ABB RobotStudio station: ProjectAPM.rsstnx

Station ProjectAPM (saved by RobotStudio 26.2.11700.0)
Controller Controller460, task T_ROB1: task frame (RAPID world) sits at (200, 0, 1400) mm in the station
Controller Controller460
  mechanical unit ROB_1: IRB460_110_240__01, 6 joints, base frame (0, 0, 0) mm
Layout (positions relative to the parent item):
  - IRB460_110_240__01 [mechanism, from %ABB.RobotStudio.Models.IRB460%\IRB460_110_240__02.rslib] at (200, 0, 1400) mm; joint values [-0.2198, 0.4757, -0.3433, 0.02] (rad or m)
  - SC_PM_PLC [smart component, from %AD3BFF28-CFC8-4A83-9FC3-1BF366785115%\SC_PM_PLC.rslib]
      properties: SimulationQuickStart=; StatisticsInfo=; con0_ID={755c8d52-c703-4704-be43-8eb584e27281}; con0_pmPLC_dpSelectedFlowID=; con0_T_ROB1_ID={f23f62ef-cbdf-4f0c-95f8-80ade90c0930}; con0_T_ROB1_ObjectReleased=(none)
  - PalletDispenser 1300_1300_300 [smart component, from %567FE6EA-F242-46D1-87E8-57A1ECE2G0DC%\PalletDispenser 1300_1300_300.rslib] at (2250, -5860, 70) mm, rotated rx 0 ry 0 rz 90 deg
      properties: PreparationTime_ToPick=0; Product_ToPick=; ClearTime_Placed=0; Product_Placed=
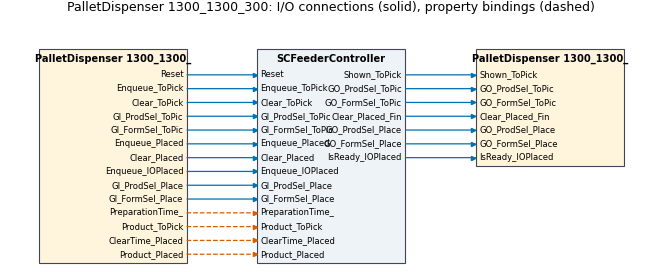
      connections:
        PalletDispenser 1300_1300_300.Reset -> SCFeederController.Reset
        PalletDispenser 1300_1300_300.Enqueue_ToPick -> SCFeederController.Enqueue_ToPick
        SCFeederController.Shown_ToPick -> PalletDispenser 1300_1300_300.Shown_ToPick
        PalletDispenser 1300_1300_300.Clear_ToPick -> SCFeederController.Clear_ToPick
        PalletDispenser 1300_1300_300.GI_ProdSel_ToPick -> SCFeederController.GI_ProdSel_ToPick
        PalletDispenser 1300_1300_300.GI_FormSel_ToPick -> SCFeederController.GI_FormSel_ToPick
        SCFeederController.GO_ProdSel_ToPick -> PalletDispenser 1300_1300_300.GO_ProdSel_ToPick
        SCFeederController.GO_FormSel_ToPick -> PalletDispenser 1300_1300_300.GO_FormSel_ToPick
        SCFeederController.Clear_Placed_Finished -> PalletDispenser 1300_1300_300.Clear_Placed_Finished
        PalletDispenser 1300_1300_300.Enqueue_Placed -> SCFeederController.Enqueue_Placed
        PalletDispenser 1300_1300_300.Clear_Placed -> SCFeederController.Clear_Placed
        PalletDispenser 1300_1300_300.Enqueue_IOPlacedRequest -> SCFeederController.Enqueue_IOPlacedRequest
        PalletDispenser 1300_1300_300.GI_ProdSel_PlacedRequest -> SCFeederController.GI_ProdSel_PlacedRequest
        PalletDispenser 1300_1300_300.GI_FormSel_PlacedRequest -> SCFeederController.GI_FormSel_PlacedRequest
        SCFeederController.GO_ProdSel_PlacedRequest -> PalletDispenser 1300_1300_300.GO_ProdSel_PlacedRequest
        SCFeederController.GO_FormSel_PlacedRequest -> PalletDispenser 1300_1300_300.GO_FormSel_PlacedRequest
        SCFeederController.IsReady_IOPlacedRequest -> PalletDispenser 1300_1300_300.IsReady_IOPlacedRequest
        PalletDispenser 1300_1300_300.PreparationTime_ToPick => SCFeederController.PreparationTime_ToPick
        PalletDispenser 1300_1300_300.Product_ToPick => SCFeederController.Product_ToPick
        PalletDispenser 1300_1300_300.ClearTime_Placed => SCFeederController.ClearTime_Placed
        PalletDispenser 1300_1300_300.Product_Placed => SCFeederController.Product_Placed
    - PalletDispenser 1300_1300_300 [part, from %567FE6EA-F242-46D1-87E8-57A1ECE2G0DC%\PalletDispenser 1300_1300_300.rslib]
    - SCFeederController [smart component, from %AD3BFF28-CFC8-4A83-9FC3-1BF366785115%\SC_FeederController.rslib]
        properties: Product_Placed=12; ClearTime_Placed=0; PreparationTime_ToPick=0; Product_ToPick=12
  - SC_Conveyor600 [smart component]
  - SixPackComponent [smart component]
      signals: DI Start, DI Pieza, DO PosicionAg
      connections:
        Source_2.Executed -> LogicSRLatch.Set
        LogicSRLatch.Output -> LinearMover.Execute
        Source_3.Executed -> LogicSRLatch_2.Set
        LogicSRLatch_2.Output -> LinearMover.Execute
        LineSensor.SensorOut -> LogicGate.InputA
        SixPackComponent.Start -> LogicGate.InputB
        LogicGate.Output -> Source_3.Execute
        LineSensor.SensorOut -> Source_3.Execute
        LogicGate_2.Output -> Source_3.Execute
        SixPackComponent.Start -> LogicGate_4.InputA
        LogicGate_4.Output -> LogicGate_2.InputA
        SixPackComponent.Pieza -> LogicGate_4.InputB
        LogicGate_4.Output -> Source_3.Execute
        LineSensor_4.SensorOut -> LogicSRLatch_2.Reset
        SixPackComponent.Start -> Source_4.Execute
        Source_3.Copy => LinearMover.Object
    - SixPack [part] at (0, 3800, 165.66) mm, rotated rx 90 ry 0 rz 0 deg, size 377 x 385.4 x 237.4 mm
    - Conveyor_600 [smart component, from %567FE6EA-F242-46D1-87E8-57A1ECE2G0DC%\Conveyor_600.rslib] at (350, 1000, 0) mm, rotated rx 0 ry 0 rz 90 deg
        properties: PreparationTime_ToPick=0; Product_ToPick=; ClearTime_Placed=0; Product_Placed=
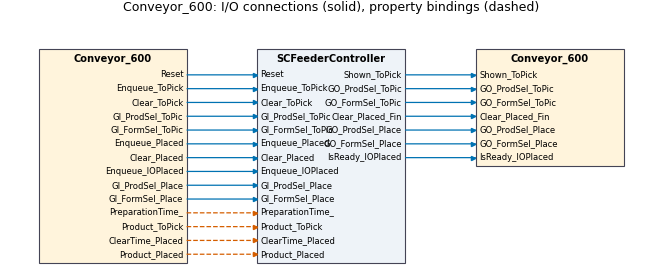
        connections:
          Conveyor_600.Reset -> SCFeederController.Reset
          Conveyor_600.Enqueue_ToPick -> SCFeederController.Enqueue_ToPick
          SCFeederController.Shown_ToPick -> Conveyor_600.Shown_ToPick
          Conveyor_600.Clear_ToPick -> SCFeederController.Clear_ToPick
          Conveyor_600.GI_ProdSel_ToPick -> SCFeederController.GI_ProdSel_ToPick
          Conveyor_600.GI_FormSel_ToPick -> SCFeederController.GI_FormSel_ToPick
          SCFeederController.GO_ProdSel_ToPick -> Conveyor_600.GO_ProdSel_ToPick
          SCFeederController.GO_FormSel_ToPick -> Conveyor_600.GO_FormSel_ToPick
          SCFeederController.Clear_Placed_Finished -> Conveyor_600.Clear_Placed_Finished
          Conveyor_600.Enqueue_Placed -> SCFeederController.Enqueue_Placed
          Conveyor_600.Clear_Placed -> SCFeederController.Clear_Placed
          Conveyor_600.Enqueue_IOPlacedRequest -> SCFeederController.Enqueue_IOPlacedRequest
          Conveyor_600.GI_ProdSel_PlacedRequest -> SCFeederController.GI_ProdSel_PlacedRequest
          Conveyor_600.GI_FormSel_PlacedRequest -> SCFeederController.GI_FormSel_PlacedRequest
          SCFeederController.GO_ProdSel_PlacedRequest -> Conveyor_600.GO_ProdSel_PlacedRequest
          SCFeederController.GO_FormSel_PlacedRequest -> Conveyor_600.GO_FormSel_PlacedRequest
          SCFeederController.IsReady_IOPlacedRequest -> Conveyor_600.IsReady_IOPlacedRequest
          Conveyor_600.PreparationTime_ToPick => SCFeederController.PreparationTime_ToPick
          Conveyor_600.Product_ToPick => SCFeederController.Product_ToPick
          Conveyor_600.ClearTime_Placed => SCFeederController.ClearTime_Placed
          Conveyor_600.Product_Placed => SCFeederController.Product_Placed
      - 600_guide [part, from %567FE6EA-F242-46D1-87E8-57A1ECE2G0DC%\Conveyor_600.rslib]
      - SCFeederController [smart component, from %AD3BFF28-CFC8-4A83-9FC3-1BF366785115%\SC_FeederController.rslib]
          properties: Product_Placed=; ClearTime_Placed=0; PreparationTime_ToPick=0; Product_ToPick=
    - LinearMover [smart component, from Components\LinearMover.rslib]
        properties: Object=(none); Direction=[0 -1 0]; Speed=5; Reference=Global; ReferenceObject=(none)
    - Source_3 [smart component, from Components\Source.rslib]
        properties: Source=SixPack; Copy=(none); Parent=(none); Position=[0 3.8000000000000003 0.96]; Orientation=[1.5707963267948966 -0 0]; Transient=true; PhysicsBehavior=0
    - LogicSRLatch_2 [smart component, from Components\LogicSRLatch.rslib]
    - LineSensor_4 [smart component, from Components\LineSensor.rslib]
        properties: Start=[0.35000000000000003 1.3 0.85]; End=[-0.29 1.3 0.85]; Length=0.64; Radius=0; Tag=(none); SenseMultiple=false; SensedPart=(none); SensedPoint=[0 0 0]
      - _sensorPart_ [part], size 640 x 0 x 0 mm
    - LogicGate_4 [smart component, from Components\LogicGate.rslib]
        properties: Operator=OR; Delay=0
    - Source_4 [smart component, from Components\Source.rslib]
        properties: Source=slipSheet; Copy=(none); Parent=(none); Position=[-1.3 -2 0.4]; Orientation=[0 0 0]; Transient=true; PhysicsBehavior=0
    - SixPack_65 [part] at (0, 3800, 960) mm, rotated rx 90 ry 0 rz 0 deg, size 377 x 385.4 x 237.4 mm
    - SixPack_171 [part] at (0, 3800, 960) mm, rotated rx 90 ry 0 rz 0 deg, size 377 x 385.4 x 237.4 mm
    - SixPack_349 [part] at (0, 3800, 960) mm, rotated rx 90 ry 0 rz 0 deg, size 377 x 385.4 x 237.4 mm
  - Grashping [smart component]
      signals: DI Atach, DI Detatch
      connections:
        LineSensor_10.SensorOut -> Attacher.Execute
        Grashping.Atach -> LogicGate_3.InputA
        LogicGate_3.Output -> Detacher.Execute
        Grashping.Atach -> LineSensor_10.Active
        Grashping.Detatch -> Detacher.Execute
        Grashping.Atach -> LineSensor_11.Active
        LineSensor_11.SensorOut -> Attacher.Execute
        Grashping.Detatch -> Attacher_2.Execute
        Grashping.Detatch -> LineSensor_3.Active
        LineSensor_10.SensedPart => Attacher.Child
        Attacher.Child => Detacher.Child
        LineSensor_11.SensedPart => Attacher.Child
        Attacher.Child => Attacher_2.Child
        LineSensor_3.SensedPart => Attacher_2.Parent
    - Attacher [smart component, from Components\Attacher.rslib]
        properties: Parent=ClampOneZoneGripper; Flange=0; Child=(none); Mount=false; Offset=[0 0 0]; Orientation=[0 0 0]
    - Detacher [smart component, from Components\Detacher.rslib]
        properties: Child=(none); KeepPosition=true
    - ClampOneZoneGripper [smart component, from %8E81373A-26AF-41AD-988A-D568DD9CCF0C%\ClampOneZoneGripper.rslib] at (1705, 0, 2836) mm, rotated rx 180 ry 0 rz 180 deg
        properties: ReleasedObject=(none)
        connections:
          ClampOneZoneGripper.giOpenClamp -> Clamp1.giOpenClamp
          Clamp1.goClampOpened -> ClampOneZoneGripper.goClampOpened
          ClampOneZoneGripper.giOpenHook -> Clamp1.giOpenHook
          Clamp1.goHookOpened -> ClampOneZoneGripper.goHookOpened
          Clamp1.doObjectReleased -> Gripper_SCPropertiesMulti2Single.DI0
          Gripper_SCPropertiesMulti2Single.DO -> ClampOneZoneGripper.doObjectReleased
          Clamp1.ReleasedObject => Gripper_SCPropertiesMulti2Single.PI0
          Gripper_SCPropertiesMulti2Single.PO => ClampOneZoneGripper.ReleasedObject
      - ClampOneZoneGripper [mechanism, from %8E81373A-26AF-41AD-988A-D568DD9CCF0C%\ClampOneZoneGripper.rslib] at (0, 0, 0) mm; joint values [0.03, 0.085, -0.0436] (rad or m)
      - Clamp1 [smart component]
          properties: ReleasedObject=(none)
          signals: GI giOpenClamp, GO goClampOpened, GI giOpenHook, GO goHookOpened, DO doObjectReleased
          connections:
            Clamp1.giOpenClamp -> ClampControl.giOpenClamp
            ClampControl.goClampOpened -> Clamp1.goClampOpened
            Clamp1.giOpenHook -> HookControl.giOpenHook
            HookControl.goHookOpened -> Clamp1.goHookOpened
            ClampAct.doObjectDetached -> Clamp1.doObjectReleased
            ClampControl.Closed -> LogicSRLatch.Set
            ClampControl.Opening -> LogicSRLatch.Reset
            LogicSRLatch.Output -> ClampAct.diAttachOrDetach
            ClampControl.Closed -> LogicGate.InputA
            ClampControl.Opening -> LogicGate.InputB
            LogicGate.Output -> ClampAct.Active
            ClampAct.ReleasedObject => Clamp1.ReleasedObject
        - ClampControl [smart component]
            signals: GI giOpenClamp, GO goClampOpened, DO Closing, DO Closed, DO Opening, DO Opened
            connections:
              JointMoverClose.Executing -> ClampControl.Closing
              JointMoverClose.Executed -> ClampControl.Closed
              JointMoverOpen.Executing -> ClampControl.Opening
              JointMoverOpen.Executed -> ClampControl.Opened
              ClampControl.giOpenClamp -> MultiSignalJudgeOpen.GI0
              MultiSignalJudgeOpen.DO -> JointMoverOpen.Execute
              JointMoverOpen.Executed -> MultiSignalSetOpen.Set
              ClampControl.giOpenClamp -> MultiSignalJudgeClose.GI0
              MultiSignalJudgeClose.DO -> JointMoverClose.Execute
              JointMoverClose.Executed -> MultiSignalSetClose.Set
              MultiSignalSetOpen.Executed -> MutiSignalSelector.SelectorA
              MultiSignalSetOpen.GO0 -> MutiSignalSelector.GiA0
              MultiSignalSetClose.Executed -> MutiSignalSelector.SelectorB
              MultiSignalSetClose.GO0 -> MutiSignalSelector.GiB0
              MutiSignalSelector.goClampOpened -> ClampControl.goClampOpened
          - MultiSignalJudgeOpen [smart component, from %AD3BFF28-CFC8-4A83-9FC3-1BF366785115%\SC_MultiSignalJudge.rslib]
              properties: DICount=0; GICount=1
          - JointMoverOpen [smart component, from %AD3BFF28-CFC8-4A83-9FC3-1BF366785115%\SC_JointMoverEx.rslib]
              properties: Mechanism=ClampOneZoneGripper; Relative=false; Duration=0.2; UseJ1=false; J1=0; UseJ2=true; J2=0; UseJ3=false; J3=0
          - MultiSignalSetOpen [smart component, from %AD3BFF28-CFC8-4A83-9FC3-1BF366785115%\SC_MultiSignalSet.rslib]
              properties: DOCount=0; GOCount=1
          - MultiSignalJudgeClose [smart component, from %AD3BFF28-CFC8-4A83-9FC3-1BF366785115%\SC_MultiSignalJudge.rslib]
              properties: DICount=0; GICount=1
          - JointMoverClose [smart component, from %AD3BFF28-CFC8-4A83-9FC3-1BF366785115%\SC_JointMoverEx.rslib]
              properties: Mechanism=ClampOneZoneGripper; Relative=false; Duration=0.2; UseJ1=false; J1=0; UseJ2=true; J2=0.085; UseJ3=false; J3=0
          - MultiSignalSetClose [smart component, from %AD3BFF28-CFC8-4A83-9FC3-1BF366785115%\SC_MultiSignalSet.rslib]
              properties: DOCount=0; GOCount=1
          - MutiSignalSelector [smart component, from %AD3BFF28-CFC8-4A83-9FC3-1BF366785115%\SC_MultiSignalSelector.rslib]
              properties: DICountA=0; GICountA=1; DICountB=0; GICountB=1; PiGiA0=goClampOpened; PiGiB0=goClampOpened
        - HookControl [smart component]
            signals: GI giOpenHook, GO goHookOpened, DO Closing, DO Closed, DO Opening, DO Opened
            connections:
              JointMoverClose.Executing -> HookControl.Closing
              JointMoverClose.Executed -> HookControl.Closed
              JointMoverOpen.Executing -> HookControl.Opening
              JointMoverOpen.Executed -> HookControl.Opened
              HookControl.giOpenHook -> MultiSignalJudgeOpen.GI0
              MultiSignalJudgeOpen.DO -> JointMoverOpen.Execute
              JointMoverOpen.Executed -> MultiSignalSetOpen.Set
              HookControl.giOpenHook -> MultiSignalJudgeClose.GI0
              MultiSignalJudgeClose.DO -> JointMoverClose.Execute
              JointMoverClose.Executed -> MultiSignalSetClose.Set
              MultiSignalSetOpen.Executed -> MutiSignalSelector.SelectorA
              MultiSignalSetOpen.GO0 -> MutiSignalSelector.GiA0
              MultiSignalSetClose.Executed -> MutiSignalSelector.SelectorB
              MultiSignalSetClose.GO0 -> MutiSignalSelector.GiB0
              MutiSignalSelector.goHookOpened -> HookControl.goHookOpened
          - MultiSignalJudgeOpen [smart component, from %AD3BFF28-CFC8-4A83-9FC3-1BF366785115%\SC_MultiSignalJudge.rslib]
              properties: DICount=0; GICount=1
          - JointMoverOpen [smart component, from %AD3BFF28-CFC8-4A83-9FC3-1BF366785115%\SC_JointMoverEx.rslib]
              properties: Mechanism=ClampOneZoneGripper; Relative=false; Duration=0.2; UseJ1=false; J1=0; UseJ2=false; J2=0; UseJ3=true; J3=1.30899693899575
          - MultiSignalSetOpen [smart component, from %AD3BFF28-CFC8-4A83-9FC3-1BF366785115%\SC_MultiSignalSet.rslib]
              properties: DOCount=0; GOCount=1
          - MultiSignalJudgeClose [smart component, from %AD3BFF28-CFC8-4A83-9FC3-1BF366785115%\SC_MultiSignalJudge.rslib]
              properties: DICount=0; GICount=1
          - JointMoverClose [smart component, from %AD3BFF28-CFC8-4A83-9FC3-1BF366785115%\SC_JointMoverEx.rslib]
              properties: Mechanism=ClampOneZoneGripper; Relative=false; Duration=0.2; UseJ1=false; J1=0; UseJ2=false; J2=0; UseJ3=true; J3=-0.0436332312998582
          - MultiSignalSetClose [smart component, from %AD3BFF28-CFC8-4A83-9FC3-1BF366785115%\SC_MultiSignalSet.rslib]
              properties: DOCount=0; GOCount=1
          - MutiSignalSelector [smart component, from %AD3BFF28-CFC8-4A83-9FC3-1BF366785115%\SC_MultiSignalSelector.rslib]
              properties: DICountA=0; GICountA=1; DICountB=0; GICountB=1; PiGiA0=goHookOpened; PiGiB0=goHookOpened
        - ClampAct [smart component] at (0, 0, 323) mm
            properties: ReleasedObject=(none); AttachedObject=(none)
            signals: DI diAttachOrDetach, DI Active, DO doObjectAttached, DO doObjectDetached
            connections:
              ClampAct.diAttachOrDetach -> SC_VolumeGripper.AttachOrDetach
              SC_VolumeGripper.TriggerAttach -> Attacher.Execute
              SC_VolumeGripper.TriggerDetach -> Detacher.Execute
              Attacher.Executed -> ClampAct.doObjectAttached
              Detacher.Executed -> ClampAct.doObjectDetached
              ClampAct.Active -> SC_VolumeGripper.Active
              SC_VolumeGripper.AttachParent => Attacher.Parent
              SC_VolumeGripper.ChildToAttach => Attacher.Child
              SC_VolumeGripper.AttachedChild => Detacher.Child
              SC_VolumeGripper.AttachedChild => ClampAct.AttachedObject
              SC_VolumeGripper.ReleasedChild => ClampAct.ReleasedObject
          - SC_VolumeGripper [smart component, from %AD3BFF28-CFC8-4A83-9FC3-1BF366785115%\SC_VolumeGripper.rslib]
              properties: Position=[0 0 0]; Orientation=[0 0 0]; Size=[0.2 0.2 0.4]; AttachParent=ClampAct; ChildToAttach=(none); AttachedChild=(none); ReleasedChild=(none)
            - _sensorPart_ [part] at (-801.98, -408.83, 179.7) mm, rotated rx 0 ry 0 rz -55.45 deg, size 200 x 200 x 400 mm
          - Attacher [smart component, from Components\Attacher.rslib]
              properties: Parent=ClampAct; Flange=0; Child=(none); Mount=false; Offset=[0 0 0]; Orientation=[0 0 0]
          - Detacher [smart component, from Components\Detacher.rslib]
              properties: Child=(none); KeepPosition=true
        - LogicSRLatch [smart component, from Components\LogicSRLatch.rslib]
        - LogicGate [smart component, from Components\LogicGate.rslib]
            properties: Operator=OR; Delay=0
      - Gripper_SCPropertiesMulti2Single [smart component, from %AD3BFF28-CFC8-4A83-9FC3-1BF366785115%\SC_PropertiesMulti2Single.rslib]
          properties: Count=1; PO=(none); PI0=(none)
    - LineSensor_11 [smart component, from Components\LineSensor.rslib] at (1705, 0, 2309) mm, rotated rx 180 ry 0 rz 180 deg
        properties: Start=[1.5596846730803193E-09 -9.080824692198064E-08 1.1309381164892329E-07]; End=[1.5596846730803193E-09 -9.080824692198064E-08 -0.3109998869061883]; Length=0.31099999999999994; Radius=0.02; Tag=(none); SenseMultiple=false; SensedPart=(none); SensedPoint=[0.04999999237060547 1.3559327392578124 0.82682470703125]
      - _sensorPart_ [part], size 40 x 40 x 311 mm
    - Attacher_2 [smart component, from Components\Attacher.rslib]
        properties: Parent=DWPallet; Flange=0; Child=(none); Mount=false; Offset=[0 0 0]; Orientation=[0 0 0]
    - LineSensor_3 [smart component, from Components\LineSensor.rslib]
        properties: Start=[1.1362 -0.495618 0.43707799999999997]; End=[1.370596 -0.376168 0.532328]; Length=0.27978983150929543; Radius=0.003; Tag=(none); SenseMultiple=false; SensedPart=DWPallet; SensedPoint=[1.136199951171875 -0.4956180114746094 0.4370780029296875]
      - _sensorPart_ [part], size 237.7 x 124.8 x 100.9 mm
  - SixPack [graphiccomponentgroup] at (0, 0, -2383.34) mm
    - SixPack [part] at (150, 120, 0) mm, rotated rx 90 ry 0 rz 0 deg, size 238.9 x 259.1 x 149.8 mm
    - OuterLine [part], size 380 x 240 x 380 mm
    - Labels [part]
    - Origin [part], size 78.6 x 49.5 x 382.7 mm
  - PalletCoca [graphiccomponentgroup] at (900, -500, 450) mm
    - MainBody [part], size 2280 x 1000 x 150 mm
    - OuterLine [part], size 2280 x 1000 x 150 mm
    - Labels [part]
    - Origin [part], size 456.5 x 200.5 x 151 mm
  - Pallet [smart component]
      signals: DI Finish
      connections:
        Pallet.Finish -> LinearMover.Execute
        Pallet.Finish -> LinearMover2.Execute
        LinearMover2.Executed -> Sink.Execute
        Sink.Executed -> Positioner.Execute
        Pallet.Finish -> LineSensor.Active
        LinearMover2.Executed -> Source.Execute
        Pallet.Finish -> Timer.Active
        Timer.Output -> LineSensor_2.Active
        Pallet.Finish -> LogicSRLatch.Set
        LogicSRLatch.Output -> LineSensor_2.Active
        LineSensor_2.SensorOutPulse -> LogicSRLatch.Reset
        Pallet.Finish -> Timer.Active
        Timer.Output -> LineSensor_2.Active
        LinearMover2.Object => Sink.Object
        LineSensor.SensedPart => LinearMover2.Object
        LineSensor.SensedPart => Source.Source
        LineSensor_2.SensedPart => LinearMover2.Object
        LinearMover2.Object => Source.Source
    - LinearMover2 [smart component, from Components\LinearMover2.rslib]
        properties: Object=DWPallet; Direction=[1 0 0]; Distance=2.8000000000000003; Duration=5; Reference=Global; ReferenceObject=(none)
    - Source [smart component, from Components\Source.rslib]
        properties: Source=DWPallet; Copy=(none); Parent=(none); Position=[0.06 0.01 0.4]; Orientation=[0 0 0]; Transient=true; PhysicsBehavior=0
    - LineSensor_2 [smart component, from Components\LineSensor.rslib]
        properties: Start=[1.1362 -0.495618 0.43707799999999997]; End=[2.2600000000000002 -0.376168 0.532328]; Length=1.1341372513942043; Radius=0.003; Tag=(none); SenseMultiple=false; SensedPart=DWPallet; SensedPoint=[1.136199951171875 -0.495617919921875 0.4370780029296875]
      - _sensorPart_ [part], size 1124.6 x 125.4 x 101.2 mm
    - Timer [smart component, from Components\Timer.rslib]
        properties: StartTime=0; Interval=0.5; Repeat=true; CurrentTime=0
  - PanelesD_9 [part] at (-540, -3690, 1350) mm, rotated rx 90 ry 0 rz 0 deg, size 154.4 x 1674 x 1496.8 mm
  - PanelesD_10 [part] at (-900, -2500, 1350) mm, rotated rx 90 ry 0 rz 90 deg, size 154.4 x 1674 x 1496.8 mm
  - PanelesD_11 [part] at (-2400, -2500, 1350) mm, rotated rx 90 ry 0 rz 90 deg, size 154.4 x 1674 x 1496.8 mm
  - PanelesD_13 [part] at (-3700, -2340, 1350) mm, rotated rx 90 ry 0 rz 0 deg, size 154.4 x 1674 x 1496.8 mm
  - PuertaAm [part] at (-3670, -240, 0) mm, rotated rx 90 ry 0 rz 180 deg, size 198.5 x 2020.7 x 1546 mm
  - PanelesD_14 [part] at (-3540, 2030, 1350) mm, rotated rx 90 ry 0 rz -90 deg, size 154.4 x 1674 x 1496.8 mm
  - PanelesD_15 [part] at (-2050, 2210, 1350) mm, rotated rx 90 ry 0 rz -70 deg, size 154.4 x 1674 x 1496.8 mm
  - PanelesD_16 [part] at (-3700, 730, 1350) mm, rotated rx 90 ry 0 rz 0 deg, size 154.4 x 1674 x 1496.8 mm
  - PanelesD_18 [part] at (-900, 3000, 1350) mm, rotated rx 90 ry 0 rz 0 deg, size 154.4 x 1674 x 1496.8 mm
  - PanelesD_19 [part] at (4000, 1200, 1350) mm, rotated rx 90 ry 0 rz -90 deg, size 154.4 x 1674 x 1496.8 mm
  - PanelesD_20 [part] at (2500, 1200, 1350) mm, rotated rx 90 ry 0 rz -90 deg, size 154.4 x 1674 x 1496.8 mm
  - PanelesD_21 [part] at (1290, 2090, 1350) mm, rotated rx 90 ry 0 rz -130 deg, size 154.4 x 1674 x 1496.8 mm
  - PanelesD_22 [part] at (700, 3490, 1350) mm, rotated rx 90 ry 0 rz -160 deg, size 154.4 x 1674 x 1496.8 mm
  - PanelesD_23 [part] at (600, 5000, 1350) mm, rotated rx 90 ry 0 rz 180 deg, size 154.4 x 1674 x 1496.8 mm
  - IRC5_Control-Module [part, from %ABB.RobotStudio.Models.IRC5%\IRC5_Control-Module.rslib] at (-940, 0, 100) mm, rotated rx 90 ry 0 rz -90 deg
  - Gabinete [part] at (-3000, -2780, 1000) mm, rotated rx 90 ry 0 rz -90 deg, size 261 x 610 x 400 mm
  - EmergencyPushButton [part] at (-3780, 550, 800) mm, rotated rx 0 ry -90 rz 0 deg, size 70 x 70 x 87.8 mm
  - EmergencyPushButton_8 [part] at (-3780, -1170, 800) mm, rotated rx 0 ry -90 rz 0 deg, size 70 x 70 x 87.8 mm
  - EmergencyPushButton_10 [part] at (-965, 3500, 830) mm, rotated rx 0 ry -90 rz 0 deg, size 70 x 70 x 87.8 mm
  - EmergencyPushButton_11 [part] at (3820, 1280, 1000) mm, rotated rx 0 ry -90 rz -90 deg, size 70 x 70 x 87.8 mm
  - Baliza [part] at (2230, 1360, 1800) mm, rotated rx 90 ry 0 rz 0 deg, size 53.8 x 318 x 54 mm
  - OpcUaClient_2 [smart component, from Components\OpcUaClient.rslib]
      properties: Status=Disconnected; ServerAddress=opc.tcp://localhost:62541; UseSecurity=false; AutoConnect=false; Blocking=false; Authentication=0; SignalConfiguration=NamespaceUri;IdentifierType;Identifier;ReadWrite;Signal;SignalType;Controller;Device
urn:inductiveautomation:ignition:opcua:tags;String;[default]/RSLinx_OPC/DI_Palet;Read;DI_Palet;Group;;

  - Outfeeder_1320 [smart component, from %567FE6EA-F242-46D1-87E8-57A1ECE2G0DC%\Outfeeder_1320.rslib] at (950, -700, 0) mm, rotated rx 0 ry 0 rz -90 deg
      properties: PreparationTime_ToPick=0; Product_ToPick=; ClearTime_Placed=0; Product_Placed=
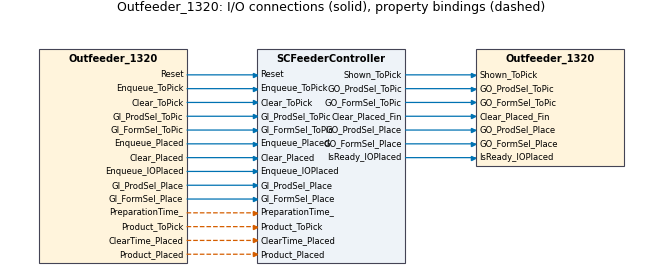
      connections:
        Outfeeder_1320.Reset -> SCFeederController.Reset
        Outfeeder_1320.Enqueue_ToPick -> SCFeederController.Enqueue_ToPick
        SCFeederController.Shown_ToPick -> Outfeeder_1320.Shown_ToPick
        Outfeeder_1320.Clear_ToPick -> SCFeederController.Clear_ToPick
        Outfeeder_1320.GI_ProdSel_ToPick -> SCFeederController.GI_ProdSel_ToPick
        Outfeeder_1320.GI_FormSel_ToPick -> SCFeederController.GI_FormSel_ToPick
        SCFeederController.GO_ProdSel_ToPick -> Outfeeder_1320.GO_ProdSel_ToPick
        SCFeederController.GO_FormSel_ToPick -> Outfeeder_1320.GO_FormSel_ToPick
        SCFeederController.Clear_Placed_Finished -> Outfeeder_1320.Clear_Placed_Finished
        Outfeeder_1320.Enqueue_Placed -> SCFeederController.Enqueue_Placed
        Outfeeder_1320.Clear_Placed -> SCFeederController.Clear_Placed
        Outfeeder_1320.Enqueue_IOPlacedRequest -> SCFeederController.Enqueue_IOPlacedRequest
        Outfeeder_1320.GI_ProdSel_PlacedRequest -> SCFeederController.GI_ProdSel_PlacedRequest
        Outfeeder_1320.GI_FormSel_PlacedRequest -> SCFeederController.GI_FormSel_PlacedRequest
        SCFeederController.GO_ProdSel_PlacedRequest -> Outfeeder_1320.GO_ProdSel_PlacedRequest
        SCFeederController.GO_FormSel_PlacedRequest -> Outfeeder_1320.GO_FormSel_PlacedRequest
        SCFeederController.IsReady_IOPlacedRequest -> Outfeeder_1320.IsReady_IOPlacedRequest
        Outfeeder_1320.PreparationTime_ToPick => SCFeederController.PreparationTime_ToPick
        Outfeeder_1320.Product_ToPick => SCFeederController.Product_ToPick
        Outfeeder_1320.ClearTime_Placed => SCFeederController.ClearTime_Placed
        Outfeeder_1320.Product_Placed => SCFeederController.Product_Placed
    - 1320_4000_h2 [part, from %567FE6EA-F242-46D1-87E8-57A1ECE2G0DC%\Outfeeder_1320.rslib]
    - SCFeederController [smart component, from %AD3BFF28-CFC8-4A83-9FC3-1BF366785115%\SC_FeederController.rslib]
        properties: Product_Placed=; ClearTime_Placed=0; PreparationTime_ToPick=0; Product_ToPick=
  - Outfeeder 1200_804 [smart component, from %567FE6EA-F242-46D1-87E8-57A1ECE2G0DC%\Outfeeder 1200_800.rslib] at (1000, -5750, 530) mm
      properties: PreparationTime_ToPick=0; Product_ToPick=; ClearTime_Placed=0; Product_Placed=
      connections:
        Outfeeder 1200_804.Reset -> SCFeederController.Reset
        Outfeeder 1200_804.Enqueue_ToPick -> SCFeederController.Enqueue_ToPick
        SCFeederController.Shown_ToPick -> Outfeeder 1200_804.Shown_ToPick
        Outfeeder 1200_804.Clear_ToPick -> SCFeederController.Clear_ToPick
        Outfeeder 1200_804.GI_ProdSel_ToPick -> SCFeederController.GI_ProdSel_ToPick
        Outfeeder 1200_804.GI_FormSel_ToPick -> SCFeederController.GI_FormSel_ToPick
        SCFeederController.GO_ProdSel_ToPick -> Outfeeder 1200_804.GO_ProdSel_ToPick
        SCFeederController.GO_FormSel_ToPick -> Outfeeder 1200_804.GO_FormSel_ToPick
        SCFeederController.Clear_Placed_Finished -> Outfeeder 1200_804.Clear_Placed_Finished
        Outfeeder 1200_804.Enqueue_Placed -> SCFeederController.Enqueue_Placed
        Outfeeder 1200_804.Clear_Placed -> SCFeederController.Clear_Placed
        Outfeeder 1200_804.Enqueue_IOPlacedRequest -> SCFeederController.Enqueue_IOPlacedRequest
        Outfeeder 1200_804.GI_ProdSel_PlacedRequest -> SCFeederController.GI_ProdSel_PlacedRequest
        Outfeeder 1200_804.GI_FormSel_PlacedRequest -> SCFeederController.GI_FormSel_PlacedRequest
        SCFeederController.GO_ProdSel_PlacedRequest -> Outfeeder 1200_804.GO_ProdSel_PlacedRequest
        SCFeederController.GO_FormSel_PlacedRequest -> Outfeeder 1200_804.GO_FormSel_PlacedRequest
        SCFeederController.IsReady_IOPlacedRequest -> Outfeeder 1200_804.IsReady_IOPlacedRequest
        Outfeeder 1200_804.PreparationTime_ToPick => SCFeederController.PreparationTime_ToPick
        Outfeeder 1200_804.Product_ToPick => SCFeederController.Product_ToPick
        Outfeeder 1200_804.ClearTime_Placed => SCFeederController.ClearTime_Placed
        Outfeeder 1200_804.Product_Placed => SCFeederController.Product_Placed
    - Pallet_Out [graphiccomponentgroup, from %567FE6EA-F242-46D1-87E8-57A1ECE2G0DC%\Outfeeder 1200_800.rslib]
      - Pallet_fixture [part, from %567FE6EA-F242-46D1-87E8-57A1ECE2G0DC%\Outfeeder 1200_800.rslib]
      - DWPallet [part, from %567FE6EA-F242-46D1-87E8-57A1ECE2G0DC%\Outfeeder 1200_800.rslib]
    - SCFeederController [smart component, from %AD3BFF28-CFC8-4A83-9FC3-1BF366785115%\SC_FeederController.rslib]
        properties: Product_Placed=; ClearTime_Placed=0; PreparationTime_ToPick=0; Product_ToPick=
  - Outfeeder 1200_805 [smart component, from %567FE6EA-F242-46D1-87E8-57A1ECE2G0DC%\Outfeeder 1200_800.rslib] at (1000, -5750, 680) mm
      properties: PreparationTime_ToPick=0; Product_ToPick=; ClearTime_Placed=0; Product_Placed=
      connections:
        Outfeeder 1200_805.Reset -> SCFeederController.Reset
        Outfeeder 1200_805.Enqueue_ToPick -> SCFeederController.Enqueue_ToPick
        SCFeederController.Shown_ToPick -> Outfeeder 1200_805.Shown_ToPick
        Outfeeder 1200_805.Clear_ToPick -> SCFeederController.Clear_ToPick
        Outfeeder 1200_805.GI_ProdSel_ToPick -> SCFeederController.GI_ProdSel_ToPick
        Outfeeder 1200_805.GI_FormSel_ToPick -> SCFeederController.GI_FormSel_ToPick
        SCFeederController.GO_ProdSel_ToPick -> Outfeeder 1200_805.GO_ProdSel_ToPick
        SCFeederController.GO_FormSel_ToPick -> Outfeeder 1200_805.GO_FormSel_ToPick
        SCFeederController.Clear_Placed_Finished -> Outfeeder 1200_805.Clear_Placed_Finished
        Outfeeder 1200_805.Enqueue_Placed -> SCFeederController.Enqueue_Placed
        Outfeeder 1200_805.Clear_Placed -> SCFeederController.Clear_Placed
        Outfeeder 1200_805.Enqueue_IOPlacedRequest -> SCFeederController.Enqueue_IOPlacedRequest
        Outfeeder 1200_805.GI_ProdSel_PlacedRequest -> SCFeederController.GI_ProdSel_PlacedRequest
        Outfeeder 1200_805.GI_FormSel_PlacedRequest -> SCFeederController.GI_FormSel_PlacedRequest
        SCFeederController.GO_ProdSel_PlacedRequest -> Outfeeder 1200_805.GO_ProdSel_PlacedRequest
        SCFeederController.GO_FormSel_PlacedRequest -> Outfeeder 1200_805.GO_FormSel_PlacedRequest
        SCFeederController.IsReady_IOPlacedRequest -> Outfeeder 1200_805.IsReady_IOPlacedRequest
        Outfeeder 1200_805.PreparationTime_ToPick => SCFeederController.PreparationTime_ToPick
        Outfeeder 1200_805.Product_ToPick => SCFeederController.Product_ToPick
        Outfeeder 1200_805.ClearTime_Placed => SCFeederController.ClearTime_Placed
        Outfeeder 1200_805.Product_Placed => SCFeederController.Product_Placed
    - Pallet_Out [graphiccomponentgroup, from %567FE6EA-F242-46D1-87E8-57A1ECE2G0DC%\Outfeeder 1200_800.rslib]
      - Pallet_fixture [part, from %567FE6EA-F242-46D1-87E8-57A1ECE2G0DC%\Outfeeder 1200_800.rslib]
      - DWPallet [part, from %567FE6EA-F242-46D1-87E8-57A1ECE2G0DC%\Outfeeder 1200_800.rslib]
    - SCFeederController [smart component, from %AD3BFF28-CFC8-4A83-9FC3-1BF366785115%\SC_FeederController.rslib]
        properties: Product_Placed=; ClearTime_Placed=0; PreparationTime_ToPick=0; Product_ToPick=
  - PanelesD_29 [part] at (-540, -5190, 1350) mm, rotated rx 90 ry 0 rz 0 deg, size 154.4 x 1674 x 1496.8 mm
  - PanelesD_33 [part] at (2960, -4210, 1350) mm, rotated rx 90 ry 0 rz 180 deg, size 154.4 x 1674 x 1496.8 mm
  - PanelesD_34 [part] at (2960, -2710, 1350) mm, rotated rx 90 ry 0 rz 180 deg, size 154.4 x 1674 x 1496.8 mm
  - PanelesD_35 [part] at (2960, -1210, 1350) mm, rotated rx 90 ry 0 rz 180 deg, size 154.4 x 1674 x 1496.8 mm
  - PanelesD_36 [part] at (600, -5510, 1350) mm, rotated rx 90 ry 0 rz 90 deg, size 154.4 x 1674 x 1496.8 mm
  - PanelesD_37 [part] at (4300, -1000, 1350) mm, rotated rx 90 ry 0 rz 90 deg, size 154.4 x 1674 x 1496.8 mm
  - Baliza_3 [part] at (-1000, 2500, 1800) mm, rotated rx 90 ry 0 rz 0 deg, size 53.8 x 318 x 54 mm
  - 48 IN LIGHT CURTAIN BODY [part] at (3700, 1200, 100) mm, rotated rx 90 ry 0 rz 0 deg, size 69.9 x 1485.9 x 57.2 mm
  - 48 IN LIGHT CURTAIN BODY_2 [part] at (3700, 520, 100) mm, rotated rx 90 ry 0 rz 180 deg, size 69.9 x 1485.9 x 57.2 mm
  - 48 IN LIGHT CURTAIN BODY_3 [part] at (-3600, 550, 100) mm, rotated rx 90 ry 0 rz 180 deg, size 69.9 x 1485.9 x 57.2 mm
  - 48 IN LIGHT CURTAIN BODY_7 [part] at (-3600, -1050, 100) mm, rotated rx 90 ry 0 rz 180 deg, size 69.9 x 1485.9 x 57.2 mm
  - 48 IN LIGHT CURTAIN BODY_8 [part] at (-880, 3500, 100) mm, rotated rx 90 ry 0 rz 90 deg, size 69.9 x 1485.9 x 57.2 mm
  - 48 IN LIGHT CURTAIN BODY_9 [part] at (-380, 3500, 100) mm, rotated rx 90 ry 0 rz 90 deg, size 69.9 x 1485.9 x 57.2 mm
  - PalletDispenser 1300_1300_301 [smart component, from %567FE6EA-F242-46D1-87E8-57A1ECE2G0DC%\PalletDispenser 1300_1300_300.rslib] at (0, -2000, 70) mm, rotated rx 0 ry 0 rz 90 deg
      properties: PreparationTime_ToPick=0; Product_ToPick=; ClearTime_Placed=0; Product_Placed=
      connections:
        PalletDispenser 1300_1300_301.Reset -> SCFeederController.Reset
        PalletDispenser 1300_1300_301.Enqueue_ToPick -> SCFeederController.Enqueue_ToPick
        SCFeederController.Shown_ToPick -> PalletDispenser 1300_1300_301.Shown_ToPick
        PalletDispenser 1300_1300_301.Clear_ToPick -> SCFeederController.Clear_ToPick
        PalletDispenser 1300_1300_301.GI_ProdSel_ToPick -> SCFeederController.GI_ProdSel_ToPick
        PalletDispenser 1300_1300_301.GI_FormSel_ToPick -> SCFeederController.GI_FormSel_ToPick
        SCFeederController.GO_ProdSel_ToPick -> PalletDispenser 1300_1300_301.GO_ProdSel_ToPick
        SCFeederController.GO_FormSel_ToPick -> PalletDispenser 1300_1300_301.GO_FormSel_ToPick
        SCFeederController.Clear_Placed_Finished -> PalletDispenser 1300_1300_301.Clear_Placed_Finished
        PalletDispenser 1300_1300_301.Enqueue_Placed -> SCFeederController.Enqueue_Placed
        PalletDispenser 1300_1300_301.Clear_Placed -> SCFeederController.Clear_Placed
        PalletDispenser 1300_1300_301.Enqueue_IOPlacedRequest -> SCFeederController.Enqueue_IOPlacedRequest
        PalletDispenser 1300_1300_301.GI_ProdSel_PlacedRequest -> SCFeederController.GI_ProdSel_PlacedRequest
        PalletDispenser 1300_1300_301.GI_FormSel_PlacedRequest -> SCFeederController.GI_FormSel_PlacedRequest
        SCFeederController.GO_ProdSel_PlacedRequest -> PalletDispenser 1300_1300_301.GO_ProdSel_PlacedRequest
        SCFeederController.GO_FormSel_PlacedRequest -> PalletDispenser 1300_1300_301.GO_FormSel_PlacedRequest
        SCFeederController.IsReady_IOPlacedRequest -> PalletDispenser 1300_1300_301.IsReady_IOPlacedRequest
        PalletDispenser 1300_1300_301.PreparationTime_ToPick => SCFeederController.PreparationTime_ToPick
        PalletDispenser 1300_1300_301.Product_ToPick => SCFeederController.Product_ToPick
        PalletDispenser 1300_1300_301.ClearTime_Placed => SCFeederController.ClearTime_Placed
        PalletDispenser 1300_1300_301.Product_Placed => SCFeederController.Product_Placed
    - PalletDispenser 1300_1300_300 [part, from %567FE6EA-F242-46D1-87E8-57A1ECE2G0DC%\PalletDispenser 1300_1300_300.rslib]
    - SCFeederController [smart component, from %AD3BFF28-CFC8-4A83-9FC3-1BF366785115%\SC_FeederController.rslib]
        properties: Product_Placed=12; ClearTime_Placed=0; PreparationTime_ToPick=0; Product_ToPick=12
  - slipSheet [part] at (1018.12, -597.6, 934.49) mm, rotated rx 0 ry 0 rz 3 deg, size 1300 x 1000 x 10 mm
  - grashping [smart component]
  - sheet_grashping [smart component]
      signals: DI Attach_sheet, DI Detach_sheet
      connections:
        LineSensor.SensorOut -> Attacher.Execute
        sheet_grashping.Attach_sheet -> LineSensor.Active
        sheet_grashping.Detach_sheet -> Detacher.Execute
        sheet_grashping.Detach_sheet -> Attacher_2.Execute
        sheet_grashping.Detach_sheet -> LineSensor_2.Active
        LineSensor.SensedPart => Attacher.Child
        Attacher.Child => Detacher.Child
        Attacher.Child => Attacher_2.Child
        LineSensor_2.SensedPart => Attacher_2.Parent
    - LineSensor [smart component, from Components\LineSensor.rslib]
        properties: Start=[0 -2 0.4]; End=[-1.3 -1 0.41000000000000003]; Length=1.6401524319403975; Radius=0.005; Tag=(none); SenseMultiple=false; SensedPart=(none); SensedPoint=[-0.7332039794921875 -1.42022705078125 0.4]
      - _sensorPart_ [part], size 1306.1 x 1007.9 x 20 mm
    - Attacher [smart component, from Components\Attacher.rslib]
        properties: Parent=ClampOneZoneGripper; Flange=0; Child=(none); Mount=false; Offset=[0 0 0]; Orientation=[0 0 0]
    - Detacher [smart component, from Components\Detacher.rslib]
        properties: Child=(none); KeepPosition=true
    - Attacher_2 [smart component, from Components\Attacher.rslib]
        properties: Parent=DWPallet; Flange=0; Child=(none); Mount=false; Offset=[0 0 0]; Orientation=[0 0 0]
    - LineSensor_2 [smart component, from Components\LineSensor.rslib]
        properties: Start=[1.1362 -0.495618 0.43707799999999997]; End=[1.370596 -0.398393 0.532328]; Length=0.27104750126315486; Radius=0.003; Tag=(none); SenseMultiple=false; SensedPart=DWPallet; SensedPoint=[1.136199951171875 -0.4956180114746094 0.4370780029296875]
      - _sensorPart_ [part], size 237.4 x 102.8 x 100.9 mm
  - Conveyor_1200_with Pallet_2 [smart component, from %567FE6EA-F242-46D1-87E8-57A1ECE2G0DC%\Conveyor_1200_with Pallet.rslib] at (1000, -500, 0) mm
      properties: PreparationTime_ToPick=0; Product_ToPick=; ClearTime_Placed=0; Product_Placed=
      connections:
        Conveyor_1200_with Pallet_2.Reset -> SCFeederController.Reset
        Conveyor_1200_with Pallet_2.Enqueue_ToPick -> SCFeederController.Enqueue_ToPick
        SCFeederController.Shown_ToPick -> Conveyor_1200_with Pallet_2.Shown_ToPick
        Conveyor_1200_with Pallet_2.Clear_ToPick -> SCFeederController.Clear_ToPick
        Conveyor_1200_with Pallet_2.GI_ProdSel_ToPick -> SCFeederController.GI_ProdSel_ToPick
        Conveyor_1200_with Pallet_2.GI_FormSel_ToPick -> SCFeederController.GI_FormSel_ToPick
        SCFeederController.GO_ProdSel_ToPick -> Conveyor_1200_with Pallet_2.GO_ProdSel_ToPick
        SCFeederController.GO_FormSel_ToPick -> Conveyor_1200_with Pallet_2.GO_FormSel_ToPick
        SCFeederController.Clear_Placed_Finished -> Conveyor_1200_with Pallet_2.Clear_Placed_Finished
        Conveyor_1200_with Pallet_2.Enqueue_Placed -> SCFeederController.Enqueue_Placed
        Conveyor_1200_with Pallet_2.Clear_Placed -> SCFeederController.Clear_Placed
        Conveyor_1200_with Pallet_2.Enqueue_IOPlacedRequest -> SCFeederController.Enqueue_IOPlacedRequest
        Conveyor_1200_with Pallet_2.GI_ProdSel_PlacedRequest -> SCFeederController.GI_ProdSel_PlacedRequest
        Conveyor_1200_with Pallet_2.GI_FormSel_PlacedRequest -> SCFeederController.GI_FormSel_PlacedRequest
        SCFeederController.GO_ProdSel_PlacedRequest -> Conveyor_1200_with Pallet_2.GO_ProdSel_PlacedRequest
        SCFeederController.GO_FormSel_PlacedRequest -> Conveyor_1200_with Pallet_2.GO_FormSel_PlacedRequest
        SCFeederController.IsReady_IOPlacedRequest -> Conveyor_1200_with Pallet_2.IsReady_IOPlacedRequest
        Conveyor_1200_with Pallet_2.PreparationTime_ToPick => SCFeederController.PreparationTime_ToPick
        Conveyor_1200_with Pallet_2.Product_ToPick => SCFeederController.Product_ToPick
        Conveyor_1200_with Pallet_2.ClearTime_Placed => SCFeederController.ClearTime_Placed
        Conveyor_1200_with Pallet_2.Product_Placed => SCFeederController.Product_Placed
    - Conv_Pallet [graphiccomponentgroup, from %567FE6EA-F242-46D1-87E8-57A1ECE2G0DC%\Conveyor_1200_with Pallet.rslib]
      - Conv_950_4000 [part, from %567FE6EA-F242-46D1-87E8-57A1ECE2G0DC%\Conveyor_1200_with Pallet.rslib]
      - DWPallet [part, from %567FE6EA-F242-46D1-87E8-57A1ECE2G0DC%\Conveyor_1200_with Pallet.rslib] at (60, 4.38, 413.27) mm
    - SCFeederController [smart component, from %AD3BFF28-CFC8-4A83-9FC3-1BF366785115%\SC_FeederController.rslib]
        properties: Product_Placed=; ClearTime_Placed=0; PreparationTime_ToPick=0; Product_ToPick=
  - slipSheet_172 [part] at (-1300, -2000, 400) mm, size 1300 x 1000 x 10 mm
  - slipSheet_350 [part] at (-1300, -2000, 400) mm, size 1300 x 1000 x 10 mm
  - Pedestal [part], size 1200 x 1000 x 1400 mm
Attachment: ClampOneZoneGripper is attached to IRB460_110_240__01 / Link6
Attachment: LineSensor_11 is attached to ClampOneZoneGripper / Base
Attachment: ? is attached to DWPallet
Attachment: ? is attached to DWPallet
Attachment: ? is attached to DWPallet
Attachment: ? is attached to DWPallet
Attachment: ? is attached to DWPallet
Attachment: ? is attached to DWPallet
Attachment: ? is attached to DWPallet
Attachment: ? is attached to DWPallet
Attachment: ? is attached to DWPallet
Attachment: ? is attached to DWPallet
Attachment: ? is attached to DWPallet
Attachment: ? is attached to DWPallet
Attachment: ? is attached to DWPallet
Attachment: ? is attached to DWPallet
Attachment: ? is attached to DWPallet
Attachment: ? is attached to DWPallet
Attachment: ? is attached to DWPallet
Attachment: ? is attached to DWPallet
Station signals: DI DI_Init
Station logic (signal -> signal, property => property):
  Controller460.pmSystem_doCycleOn -> SC_PM_PLC.con0_pmPLC_diCycleOn
  Controller460.pmSystem_doMotorOn -> SC_PM_PLC.con0_pmPLC_diMotorOn
  Controller460.pmSystem_doAutoOn -> SC_PM_PLC.con0_pmPLC_diAutoOn
  Controller460.pmSystem_doRunchOk -> SC_PM_PLC.con0_pmPLC_diRunchOk
  Controller460.pmProject_goStatus -> SC_PM_PLC.con0_pmPLC_giProjectStatus
  Controller460.DO_Attatch -> Grashping.Atach
  SixPackComponent.PosicionAg -> Controller460.DI_Cinta
  Controller460.DO_Pieza -> SixPackComponent.Pieza
  Controller460.DO_Dettatch -> Grashping.Detatch
  Controller460.DO_Finish -> Pallet.Finish
  Controller460.DO_Start -> LogicGate.InputB
  LogicGate.Output -> SixPackComponent.Start
  Controller460.DO_Start -> SixPackComponent.Start
  ProjectAPM.DI_Init -> Controller460.DI_INIT
  Controller460.DO_Attatch_Sheet -> sheet_grashping.Attach_sheet
  Controller460.DO_Dettatch_Sheet -> sheet_grashping.Detach_sheet
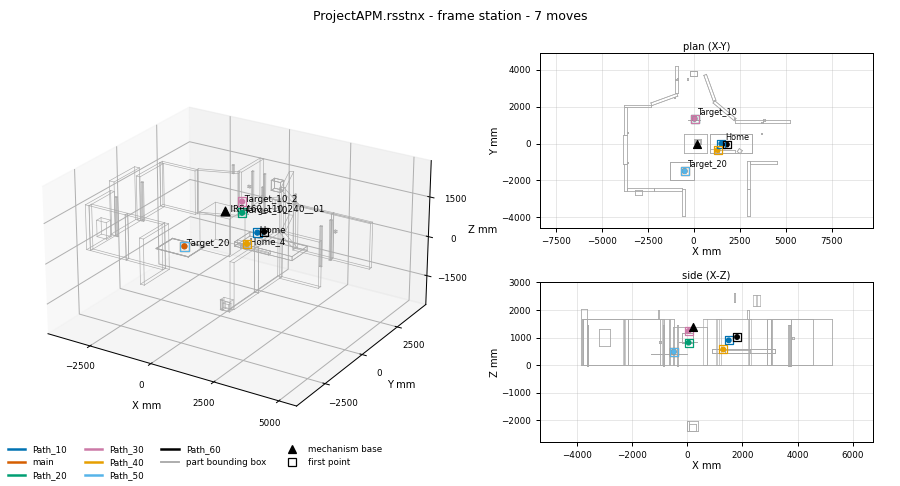
[picture p0: tool path of ProjectAPM.rsstnx in frame station, 7 of 19 moves have a stored position in this frame; points joined in program order, loops and branches not executed]
Targets, tools, work objects and paths stored in the station, written as RAPID:
! task T_ROB1
MODULE pmrcUser
  TASK PERS wobjdata pmInfeeder1_WObj:=[FALSE,TRUE,"",[[-200,0,-1400],[1,0,0,0]],[[0,0,0],[1,0,0,0]]];
  TASK PERS wobjdata pmInfeeder2_WObj:=[FALSE,TRUE,"",[[-200,0,-1400],[1,0,0,0]],[[0,0,0],[1,0,0,0]]];
  TASK PERS wobjdata pmInfeeder3_WObj:=[FALSE,TRUE,"",[[-200,0,-1400],[1,0,0,0]],[[0,0,0],[1,0,0,0]]];
  TASK PERS wobjdata pmInfeeder4_WObj:=[FALSE,TRUE,"",[[-200,0,-1400],[1,0,0,0]],[[0,0,0],[1,0,0,0]]];
  TASK PERS wobjdata pmOutfeeder1_WObj:=[FALSE,TRUE,"",[[-200,0,-1400],[1,0,0,0]],[[0,0,0],[1,0,0,0]]];
  TASK PERS wobjdata pmOutfeeder2_WObj:=[FALSE,TRUE,"",[[-200,0,-1400],[1,0,0,0]],[[0,0,0],[1,0,0,0]]];
  TASK PERS wobjdata pmOutfeeder3_WObj:=[FALSE,TRUE,"",[[-200,0,-1400],[1,0,0,0]],[[0,0,0],[1,0,0,0]]];
  TASK PERS wobjdata pmOutfeeder4_WObj:=[FALSE,TRUE,"",[[-200,0,-1400],[1,0,0,0]],[[0,0,0],[1,0,0,0]]];
  TASK PERS wobjdata pmPallet1_WObj:=[FALSE,TRUE,"",[[-200,0,-1400],[1,0,0,0]],[[0,0,0],[1,0,0,0]]];
  TASK PERS wobjdata pmSlipsheet1_WObj:=[FALSE,TRUE,"",[[-200,0,-1400],[1,0,0,0]],[[0,0,0],[1,0,0,0]]];
  TASK PERS tooldata pmPickTool1:=[TRUE,[[0,0,0],[1,0,0,0]],[1,[0,0,10],[1,0,0,0],0.01,0.01,0.01]];
  TASK PERS tooldata pmSearchTool1:=[TRUE,[[0,0,0],[1,0,0,0]],[1,[0,0,10],[1,0,0,0],0.01,0.01,0.01]];
  TASK PERS tooldata tGripper:=[TRUE,[[0,0,533],[1,0,0,0]],[45,[0,0,10],[1,0,0,0],0.609375,0.9375,0.346875]];
  TASK PERS tooldata pmCalibTool1:=[TRUE,[[0,0,0],[1,0,0,0]],[0.001,[0,0,0.001],[1,0,0,0],0,0,0]];
  PROC PmLoadReadySignalReset()
    SetDO pmSystem_doLoadReady1,0;
    SetDO pmSystem_doLoadReady2,0;
    SetDO pmSystem_doLoadReady3,0;
    SetDO pmSystem_doLoadReady4,0;
    SetDO pmSystem_doLoadReady5,0;
    SetDO pmSystem_doLoadReady6,0;
  ENDPROC
  PROC PmLoadReady()
    SetDO \Sync,pmSystem_doLoadReady1,1;
    SetDO \Sync,pmSystem_doLoadReady2,1;
    SetDO \Sync,pmSystem_doLoadReady3,1;
    SetDO \Sync,pmSystem_doLoadReady4,1;
    SetDO \Sync,pmSystem_doLoadReady5,1;
    SetDO \Sync,pmSystem_doLoadReady6,1;
  ENDPROC
  PROC PmResetProjStartFlagAtStart()
  ENDPROC
ENDMODULE

! task T_ROB1
MODULE pmrcSys
  TASK PERS wobjdata pm_home_WObj:=[FALSE,TRUE,"",[[-200,0,-1400],[1,0,0,0]],[[0,0,0],[1,0,0,0]]];
  LOCAL PERS tooldata curr_Tool:=[TRUE,[[0,0,0],[1,0,0,0]],[0.001,[0,0,0.001],[1,0,0,0],0,0,0]];
  TASK PERS tooldata PmLastTool:=[TRUE,[[0,0,0],[1,0,0,0]],[0.001,[0,0,0.001],[1,0,0,0],0,0,0]];
  LOCAL PERS wobjdata curr_WObj:=[FALSE,TRUE,"",[[-200,0,-1400],[1,0,0,0]],[[0,0,0],[1,0,0,0]]];
  TASK PERS wobjdata PmLastWobj:=[FALSE,TRUE,"",[[-200,0,-1400],[1,0,0,0]],[[0,0,0],[1,0,0,0]]];
  PROC PmSetupDummyIO()
  ENDPROC
ENDMODULE

! task T_ROB1
MODULE Module1
  CONST robtarget Target_10:=[[-150,1355.932739642,-579.936186208],[0,0,1,0],[1,0,1,0],[9E+09,9E+09,9E+09,9E+09,9E+09,9E+09]];
  CONST robtarget Home:=[[1305,0,-497],[0,0,1,0],[0,0,0,0],[9E+09,9E+09,9E+09,9E+09,9E+09,9E+09]];
  CONST robtarget Target_10_2:=[[-150,1355.932739642,-159.936186208],[0,0,1,0],[1,0,1,0],[9E+09,9E+09,9E+09,9E+09,9E+09,9E+09]];
  CONST robtarget Home_4:=[[1105,-350,-827],[0,0,1,0],[0,0,0,0],[9E+09,9E+09,9E+09,9E+09,9E+09,9E+09]];
  CONST robtarget Home_4_2:=[[1105,-350,-727],[0,0.707106781,0.707106781,0],[0,0,0,0],[9E+09,9E+09,9E+09,9E+09,9E+09,9E+09]];
  CONST robtarget Home_4_3:=[[1105,-350,-627],[0,0.707106781,0.707106781,0],[0,0,0,0],[9E+09,9E+09,9E+09,9E+09,9E+09,9E+09]];
  CONST robtarget Home_4_3_2:=[[1105,-350,-427],[0,0.707106781,0.707106781,0],[0,0,0,0],[9E+09,9E+09,9E+09,9E+09,9E+09,9E+09]];
  CONST robtarget Target_20:=[[-685.53959866,-1494.337229442,-911.485646006],[0,0.725374371,0.688354576,0],[-2,0,-1,0],[9E+09,9E+09,9E+09,9E+09,9E+09,9E+09]];
  CONST robtarget Home_4_sheet:=[[1605,-50,-377],[0,0.707106781,0.707106781,0],[0,0,0,0],[9E+09,9E+09,9E+09,9E+09,9E+09,9E+09]];
  PROC Path_10()
    MoveL Home,v7000,z10,tGripper\WObj:=wobj0;
  ENDPROC
  PROC main()
    Reset DO_Start;
    Reset DO_Pieza;
    Reset DO_Attatch;
    Reset DO_Dettatch;
    Reset DO_Attatch_Sheet;
    Reset DO_Dettatch_Sheet;
    Path_10;
    Reset DO_Dettatch_Sheet;
    Set DO_Start;
    WaitTime 0.1;
    Reset DO_Start;
    Path_30;
    Path_20;
    WaitTime 1;
    Set DO_Attatch;
    WaitTime 1;
    Path_30;
    Reset DO_Attatch;
    MoveJ palletposa,v7000,fine,tGripper\WObj:=wobj0;
    MoveL palletposa,v7000,fine,tGripper\WObj:=wobj0;
    WaitTime 0.5;
    Set DO_Dettatch;
    WaitTime 0.5;
    MoveL palletposa,v7000,fine,tGripper\WObj:=wobj0;
    Reset DO_Dettatch;
    Set DO_Start;
    WaitTime 0.1;
    Reset DO_Start;
    Path_30;
    Path_20;
    WaitTime 1;
    Set DO_Attatch;
    WaitTime 1;
    Path_30;
    Reset DO_Attatch;
    MoveJ palletposa,v7000,fine,tGripper\WObj:=wobj0;
    MoveL palletposa,v7000,fine,tGripper\WObj:=wobj0;
    WaitTime 0.5;
    Set DO_Dettatch;
    WaitTime 0.5;
    MoveL palletposa,v7000,fine,tGripper\WObj:=wobj0;
    Reset DO_Dettatch;
    Set DO_Start;
    WaitTime 0.1;
    Reset DO_Start;
    Path_30;
    Path_20;
    WaitTime 1;
    Set DO_Attatch;
    WaitTime 1;
    Path_30;
    Reset DO_Attatch;
    MoveJ palletposa,v7000,fine,tGripper\WObj:=wobj0;
    MoveJ palletposa,v7000,fine,tGripper\WObj:=wobj0;
    WaitTime 0.5;
    Set DO_Dettatch;
    WaitTime 0.5;
    MoveL palletposa,v7000,fine,tGripper\WObj:=wobj0;
    Reset DO_Dettatch;
    MoveJ pos_sheeta,v7000,fine,tGripper\WObj:=wobj0;
    MoveJ Target_20,v7000,fine,tGripper\WObj:=wobj0;
    WaitTime 1;
    Set DO_Attatch_Sheet;
    WaitTime 1;
    Reset DO_Attatch_Sheet;
    MoveJ pos_sheeta,v7000,fine,tGripper\WObj:=wobj0;
    WaitTime 1;
    MoveJ sheetpalleta,v7000,fine,tGripper\WObj:=wobj0;
    WaitTime 1;
    Set DO_Dettatch_Sheet;
    WaitTime 1;
    Set DO_Finish;
    WaitTime 1;
    Reset DO_Finish;
  ENDPROC
  PROC Path_20()
    MoveL Target_10,v7000,z10,tGripper\WObj:=wobj0;
  ENDPROC
  PROC Path_30()
    MoveJ Target_10_2,v7000,z10,tGripper\WObj:=wobj0;
  ENDPROC
  PROC Path_40()
    MoveL Home_4,v7000,z10,tGripper\WObj:=wobj0;
  ENDPROC
  PROC Path_50()
    MoveL Target_20,v7000,z100,tGripper\WObj:=wobj0;
  ENDPROC
  PROC Path_60()
    MoveL Home_4_sheet,v7000,z100,tGripper\WObj:=wobj0;
  ENDPROC
ENDMODULE

! task T_ROB1
MODULE CalibData
  TASK PERS wobjdata Paletizado:=[FALSE,TRUE,"",[[-200,0,-1400],[1,0,0,0]],[[0,0,0],[1,0,0,0]]];
ENDMODULE

